INTERFACE I_Object EXTENDS __SYSTEM.IQueryInterface

END_INTERFACE

(* stored: Version 1.1.0.1
   Itf I_Object: Id {ea8104e0-6b35-0dc0-35e1-f6e019e8e23c} *)
